{attribute 'obsolete' := 'Use E_StageBrakeMode'}
TYPE ENUM_StageBrakeMode : E_StageBrakeMode; END_TYPE

(* stored: Version 1.1.0.1
   DUT ENUM_StageBrakeMode: Id {3c0a8cbb-8e85-4a00-b022-9242db2ddeb2} *)
